(* Schneider Machine Expert - Basic project Test_Motor, file version 3.0.0.0 *)
(* ProjectInformations: Name=Test_Motor *)

HARDWARE
  Cpu 0: TM221CE24T
  EthernetConfiguration: NetworkName=M221, IpAllocationMode=ByDhcp, IpAddress=192.168.1.10, SubnetMask=255.255.255.0
  SerialLineConfiguration: Baud=Baud19200, Parity=ParityEven, DataBits=DataBits8, StopBits=StopBits1, PhysicalMedium=PhysicalMediumRs485, TransmissionMode=TransmissionModeModbusRtu, SlaveId=1, Addressing=SlaveAddressing
  MastTask: UsePeriodScanMode=false, PeriodScan=100
  FastTask: Period=255
  CpuBehavior: StartingMode=StartAsPreviousState, AutoSaveRamOnEeprom=true, WatchdogPeriod=250

SYMBOLS  (address, symbol, comment, settings)
  %M0       MTR_RUN  "Motor Running Latch"
  %I0.0     PB_START
  %I0.1     PB_STOP
  %I0.2     ESTOP
  %I0.3     OL_TRIP
  %Q0.0     MTR_OUT
  %Q0.1     LT_RUN

POU Test_Motor
  (* SectionNumber=1 *)

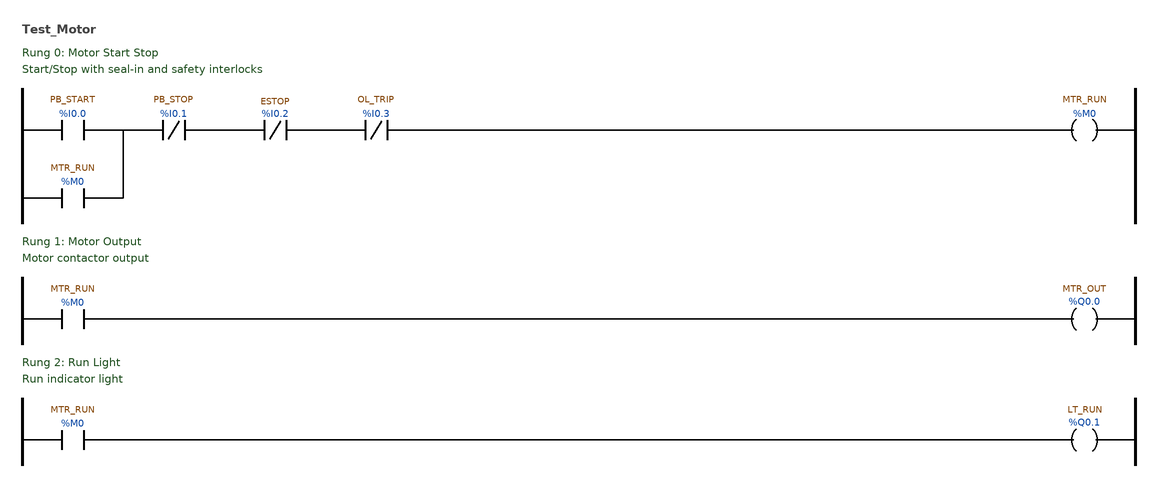

// Rung 0: Motor Start Stop
// Start/Stop with seal-in and safety interlocks
  LD %I0.0                (* PB_START *)
  OR %M0                  (* MTR_RUN *)
  ANDN %I0.1              (* PB_STOP *)
  ANDN %I0.2              (* ESTOP *)
  ANDN %I0.3              (* OL_TRIP *)
  ST %M0                  (* MTR_RUN *)
  // as ST:
  //   MTR_RUN := (PB_START OR MTR_RUN) AND NOT PB_STOP AND NOT ESTOP AND NOT OL_TRIP;

// Rung 1: Motor Output
// Motor contactor output
  LD %M0                  (* MTR_RUN *)
  ST %Q0.0                (* MTR_OUT *)
  // as ST:
  //   MTR_OUT := MTR_RUN;

// Rung 2: Run Light
// Run indicator light
  LD %M0                  (* MTR_RUN *)
  ST %Q0.1                (* LT_RUN *)
  // as ST:
  //   LT_RUN := MTR_RUN;
